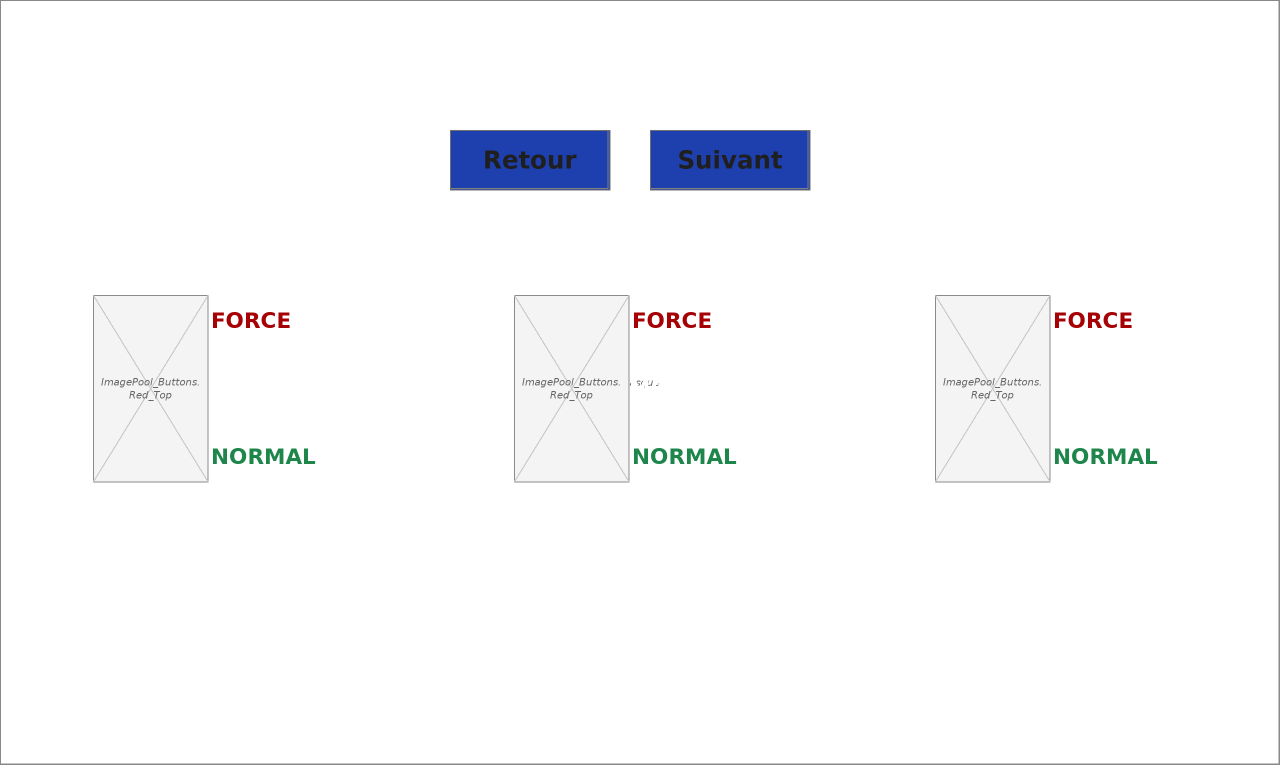
VISUALIZATION Maintenance_5  // 1280x765
    Frame (0,0 1280x765)
        shows masque()
    Button (450,130 160x60), "Retour"
        OnMouseDown: execute {
            IF (Option_WC_GV OR Option_WC_PV OR Option_Prise)
            	THEN
            	VisuElems.CURRENTVISU := 'Maintenance_4';
            	ELSIF (Option_Bas_Debit OR Option_Douchette OR Option_NEP)
            		THEN
            		VisuElems.CURRENTVISU := 'Maintenance_3';
            	ELSIF (Option_Douche OR Option_Lavabo)
            		THEN
            		VisuElems.CURRENTVISU := 'Maintenance_2';
            	ELSIF (Option_RegSouf_Ultrason OR Option_Reg_Etanche_Ext OR Option_V3V_EauMitig)
            		THEN
            		VisuElems.CURRENTVISU := 'Maintenance_1';
            	ELSE
            	VisuElems.CURRENTVISU := 'menu';
            END_IF
        }
    Button (650,130 160x60), "Suivant"
        OnMouseDown: execute {
            IF (Option_Com_RegSouf_Ultrason)
            	THEN
            		VisuElems.CURRENTVISU := 'Maintenance_6';
            	ELSE
            		VisuElems.CURRENTVISU := 'Maintenance_7';
            END_IF
        }
    Group (863,237 390x380), invisible if: NOT Option_Cabine_Climatique
        Rectangle (4,0 381x68), "Vanne Bat. froide"
        RoundedRectangle (0,244 390x68), "Ouverture : %.0f %%", text variable: F_Cons_V3V_Bat_Froid_CTA
            OnMouseDown: write the text variable via VisuDialogs.Numpad, min 0, max 100, format %.0f
        Rectangle (0,312 390x68), "Appli : %.0f %%", text variable: Cons_Actionneur_V3V_Froid_CTA
        Group (72,58 246x187)
            Group (0,0 115x187)
                Image (0,0 115x187), invisible if: EF_Cons_V3V_Bat_Froid_CTA, image: ImagePool_Buttons.Green_Bottom
                    OnMouseDown: toggle EF_Cons_V3V_Bat_Froid_CTA
                Image (0,0 115x187), invisible if: NOT EF_Cons_V3V_Bat_Froid_CTA, image: ImagePool_Buttons.Red_Top
                    OnMouseDown: toggle EF_Cons_V3V_Bat_Froid_CTA
            Rectangle (115,0 131x51), "FORCE"
            Rectangle (112,68 131x51), "MODE"
            Rectangle (115,136 131x51), "NORMAL"
    Group (21,237 390x519), invisible if: NOT Option_Cabine_Climatique
        Rectangle (4,0 381x68), "Moteur soufflage"
        RoundedRectangle (0,248 390x68), "Vitesse : %.0f %%", text variable: Tab_MotSouf_CTA.W_ConsForcage
            OnMouseDown: write the text variable via VisuDialogs.Numpad, min 0, max 100, format %.0f
        Rectangle (0,315 390x68), "Appli : %.0f %%", text variable: Tab_MotSouf_CTA.R_InfoCons
        Group (72,58 246x187)
            Group (0,0 115x187)
                Image (0,0 115x187), invisible if: Tab_MotSouf_CTA.Mot_Ecriture.0, image: ImagePool_Buttons.Green_Bottom
                    OnMouseDown: toggle Tab_MotSouf_CTA.Mot_Ecriture.0
                Image (0,0 115x187), invisible if: NOT Tab_MotSouf_CTA.Mot_Ecriture.0, image: ImagePool_Buttons.Red_Top
                    OnMouseDown: toggle Tab_MotSouf_CTA.Mot_Ecriture.0
            Rectangle (115,0 131x51), "FORCE"
            Rectangle (112,68 131x51), "MODE"
            Rectangle (115,136 131x51), "NORMAL"
        RoundedRectangle (0,383 390x68), "Vit Max : %.0f %%", text variable: Tab_MotSouf_CTA.W_LimiteMaxCons
            OnMouseDown: write the text variable via VisuDialogs.Numpad, min 0, max 100, format %.0f
        RoundedRectangle (0,451 390x68), "Vit Min : %.0f %%", text variable: Tab_MotSouf_CTA.W_LimiteMinCons
            OnMouseDown: write the text variable via VisuDialogs.Numpad, min 0, max 100, format %.0f
    Group (442,237 390x516), invisible if: NOT Option_Cabine_Climatique
        Rectangle (4,0 381x68), "Moteur reprise"
        RoundedRectangle (0,244 390x68), "Vitesse : %.0f %%", text variable: Tab_MotRep_CTA.W_ConsForcage
            OnMouseDown: write the text variable via VisuDialogs.Numpad, min 0, max 100, format %.0f
        Rectangle (0,312 390x68), "Appli : %.0f %%", text variable: Tab_MotRep_CTA.R_InfoCons
        Group (72,58 246x187)
            Group (0,0 115x187)
                Image (0,0 115x187), invisible if: Tab_MotRep_CTA.Mot_Ecriture.0, image: ImagePool_Buttons.Green_Bottom
                    OnMouseDown: toggle Tab_MotRep_CTA.Mot_Ecriture.0
                Image (0,0 115x187), invisible if: NOT Tab_MotRep_CTA.Mot_Ecriture.0, image: ImagePool_Buttons.Red_Top
                    OnMouseDown: toggle Tab_MotRep_CTA.Mot_Ecriture.0
            Rectangle (115,0 131x51), "FORCE"
            Rectangle (112,68 131x51), "MODE"
            Rectangle (115,136 131x51), "NORMAL"
        RoundedRectangle (0,448 390x68), "Vit Min : %.0f %%", text variable: Tab_MotRep_CTA.W_LimiteMinCons
            OnMouseDown: write the text variable via VisuDialogs.Numpad, min 0, max 100, format %.0f
        RoundedRectangle (0,380 390x68), "Vit Max : %.0f %%", text variable: Tab_MotRep_CTA.W_LimiteMaxCons
            OnMouseDown: write the text variable via VisuDialogs.Numpad, min 0, max 100, format %.0f
END_VISUALIZATION

(* stored: Version 1.1.0.1, ProductVersion 3.1.4024.15
   Visu Maintenance_5: Id {75c02538-757e-4723-a0b6-06e9898074cc} *)
